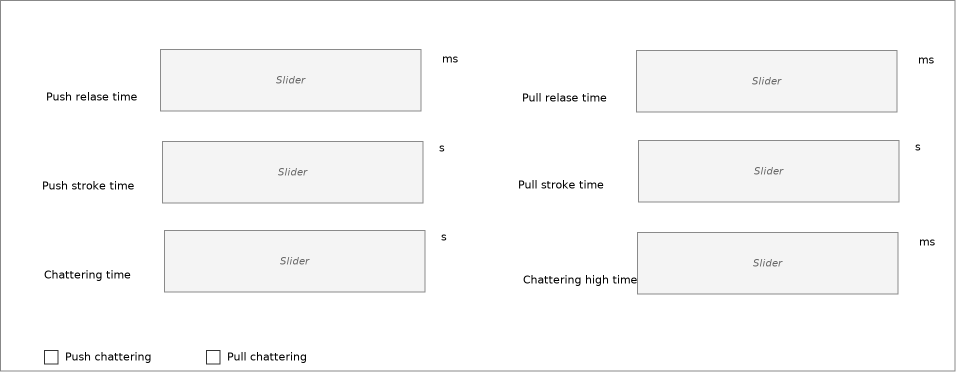
VISUALIZATION Visualization  // 956x372
    Label (43,82 150x30), "Push relase time"
    Slider (160,49 261x62), variable: SimulationMAIN.cylinder_stub.push_release_time, scale 0..1000
    Label (439,44 40x30), "ms"
    Label (519,83 150x30), "Pull relase time"
    Slider (636,50 261x62), variable: SimulationMAIN.cylinder_stub.pull_release_time, scale 0..1000
    Label (915,45 40x30), "ms"
    Slider (162,141 261x62), variable: SimulationMAIN.push_stroke_time, scale 0..10
    Label (39,171 150x30), "Push stroke time"
    Label (436,133 40x30), "s"
    Slider (638,140 261x62), variable: SimulationMAIN.pull_stroke_time, scale 0..10
    Label (515,170 150x30), "Pull stroke time"
    Label (912,132 40x30), "s"
    Slider (164,230 261x62), variable: SimulationMAIN.chattering_time, scale 0..5
    Label (41,260 150x30), "Chattering time"
    Label (438,222 40x30), "s"
    Label (520,265 150x30), "Chattering high time"
    Slider (637,232 261x62), variable: SimulationMAIN.cylinder_stub.chattering_hl_time, scale 0..100
    Label (916,227 40x30), "ms"
    Checkbox (42,342 150x30), "Push chattering", variable: SimulationMAIN.cylinder_stub.chattering_push
    Checkbox (204,342 150x30), "Pull chattering", variable: SimulationMAIN.cylinder_stub.chattering_pull
END_VISUALIZATION

(* stored: Version 1.1.0.1, ProductVersion 3.1.4024.12
   Visu Visualization: Id {3a965d44-c909-493b-8de0-64d6ababe7be} *)
